TYPE teScrewFeeders :
(
	CE_SCREW_FEED_1:=1,
	CE_SCREW_FEED_2,
	CE_SCREW_FEED_3,
	CE_SCREW_FEED_4
);
END_TYPE

(* stored: Version 1.1.0.1, ProductVersion 3.1.4022.18
   DUT teScrewFeeders: Id {afcd0368-fd89-4220-8ed4-e59648e14448} *)
